TYPE InfoDataAdsAddrStateBase_1916E49F :
STRUCT
END_STRUCT
END_TYPE

(* stored: Version 1.2.0.0, ProductVersion 3.1.4024.9
   DUT InfoDataAdsAddrStateBase_1916E49F: Id {20326140-06b9-4b38-8cf5-4bca82b9b54f} *)
